// TIA Portal V18 export
// export: Created 2026-03-12T16:04:35.0413987Z, ExportSetting WithDefaults, DisplayName Totally Integrated Automation Portal, DisplayVersion V18 Update 5, DisplayName TIA Portal Openness, DisplayVersion V18 Update 5, DisplayName TIA Portal Version Control Interface, DisplayVersion V18, DisplayName SINAMICS Startdrive Advanced, DisplayVersion V18, DisplayName SINAMICS Startdrive G130, G150, S120, S150, SINAMICS MV, S210, DisplayVersion V18, DisplayName SINAMICS Startdrive G110M, G120, G120C, G120D, G120P, G115D, DisplayVersion V18, DisplayName STEP 7 Professional, DisplayVersion V18 Update 5, DisplayName STEP 7 Safety, DisplayVersion V18, DisplayName WinCC Professional, DisplayVersion V18 Update 5
FUNCTION_BLOCK "FB SETPOINT MANUAL"   // FB14, LAD
TITLE = Function Block FB SETPOINT_MANUAL
{ S7_Optimized_Access := 'TRUE' }
VERSION : 0.1
// Cálculo de conversão do valor setado, para escala do CLP.
// stored: AutoNumber true, IsIECCheckEnabled false, IsRetainMemResEnabled false, MemoryReserve 100, SetENOAutomatically false, UDAEnableTagReadback false
   VAR_INPUT
      REMOTO : Bool;   // Recebe sinal de Remoto Manual
      COMANDO_VALOR : Int;   // Índice de comparação do bloco
      COMANDO : Int;   // Comando enviado via IHM/SCADA para definir min/max do range
      RANGE_MIN : Int;   // Valor mínimo do fundo de escala do equip, escrito via aferição
      RANGE_MAX : Int;   // Valor máximo do fundo de escala do equip, escrito via aferição
   END_VAR
   VAR_OUTPUT
      VALOR_SAIDA : Int;   // Valor de escrita no escravo.
      CADASTRO_VEL_MAX : Int;   // Cadastro da Velocidade Máxima via IHM
      CADASTRO_VEL_MIN : Int;   // Cadastro da Velocidade Mínima via IHM
   END_VAR
   VAR_IN_OUT
      SET_MANUAL : Int;   // Valor da grandeza a ser alcançado, escrita via aferição.
   END_VAR
   VAR RETAIN
      SETPOINT : Int;   // Setpoint de velocidade
      PULSE : Bool;
      PULSE_AUX : Bool;
   END_VAR
   VAR_TEMP   // added for the SCL form of the ladder/FBD networks
      _w1 : Bool;
   END_VAR
BEGIN

REGION Network 1: Cálculo Dosagem Manual
   // SET_MANUAL =  Valor da grandeza a ser alcançado, escrita via aferição.
   // RANGE_MAX   =  Valor máximo do fundo de escala do equip, escrita via aferição.
   // RANGE_MIN   =   Valor mínimo do fundo de escala do equip, escrita via aferição
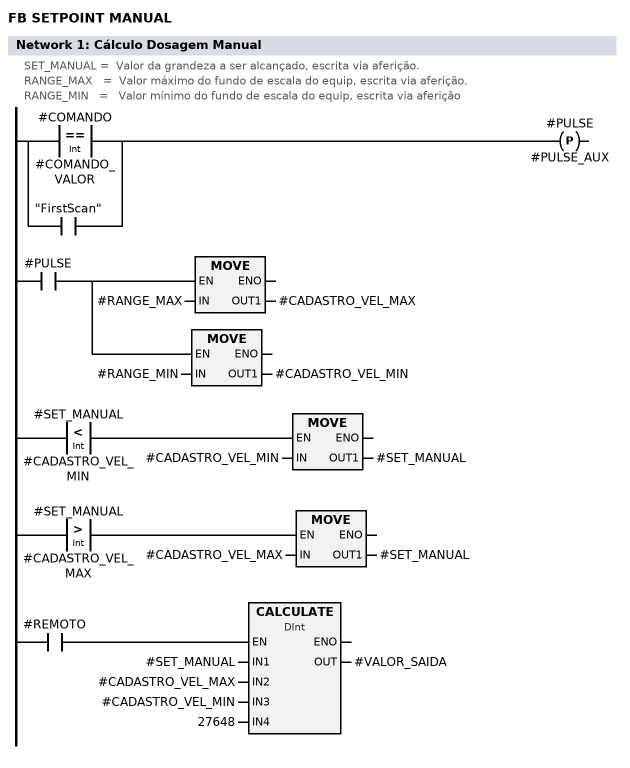
   #_w1 := (#COMANDO = #COMANDO_VALOR) OR "FirstScan";
   #PULSE := #_w1 AND NOT #PULSE_AUX;   // rising edge
   #PULSE_AUX := #_w1;
   IF #PULSE THEN
       #CADASTRO_VEL_MAX := #RANGE_MAX;
       #CADASTRO_VEL_MIN := #RANGE_MIN;
   END_IF;
   IF #SET_MANUAL < #CADASTRO_VEL_MIN THEN #SET_MANUAL := #CADASTRO_VEL_MIN; END_IF;
   IF #SET_MANUAL > #CADASTRO_VEL_MAX THEN #SET_MANUAL := #CADASTRO_VEL_MAX; END_IF;
   IF #REMOTO THEN
       #VALOR_SAIDA := ((#SET_MANUAL*27648) / (#CADASTRO_VEL_MAX-#CADASTRO_VEL_MIN)) - ((#CADASTRO_VEL_MIN*27648) / (#CADASTRO_VEL_MAX-#CADASTRO_VEL_MIN));
   END_IF;
END_REGION
END_FUNCTION_BLOCK
